TYPE ST_OPCUA_NodeVariablePair_STRING :
STRUCT
	clientVariable : STRING;
	clientVariableInfo : __SYSTEM.VAR_INFO;
	serverNodeIdentifier : STRING;
END_STRUCT
END_TYPE

(* stored: Version 1.1.0.1, ProductVersion 3.1.4024.9
   DUT ST_OPCUA_NodeVariablePair_STRING: Id {67f1656d-fead-4a2e-869f-284ae34b637e} *)
